Staubli VAL3: Control_Remote.pgx

public program Control_Remote(num& x_nMode, num& x_nCycleCount)
  local string l_sItem[2]
  local num l_nNum
  local num l_nKey
  local num l_nData[2]
  local num l_nSelectIndex
  local string l_sSMess[6]
begin

  //修改点位的 joint
  l_nData[0]=max(round(x_nMode),0)
  l_nData[1]=max(round(x_nCycleCount),0)

  l_sSMess[0]="按钮触发单工位"
  l_sSMess[1]="按钮触发单周期"
  l_sSMess[2]="按钮触发多周期"
  l_sSMess[3]="无需按钮触发"
  l_sSMess[4]="按钮触发排队"
  l_sSMess[5]="用户自定义触发"


  l_sItem[0]="生产模式:"+l_sSMess[l_nData[0]]
  l_sItem[1]="周期次数:"+toString("",l_nData[1])


  call Control_BottomS(",,,,,,取消,确定")
  call Control_PanelXY(8,0,25,2)
  call Control_ListCls()
  call Control_Panel("生产配置")
  call Control_List(l_sItem,l_nSelectIndex)
  while true
    l_nKey=getKey()

    switch l_nKey
      case 261
        l_nSelectIndex=max(0,l_nSelectIndex-1)
      break

      case 266
        l_nSelectIndex=min(l_nSelectIndex+1,1)
      break

      case 278
        x_nMode=l_nData[0]
        x_nCycleCount=l_nData[1]

        return
      break


      case 277
        return
      break

      case 270
        if l_nSelectIndex==0
         call Sel_Edit(l_nData[0],nPanelLTopX+10,nPanelLTopY+1,l_sSMess)
        else
          call Float_Edit(l_nData[1],nPanelLTopX+10,nPanelLTopY+2)

        endIf



        l_nData[l_nSelectIndex]=max(round(l_nData[l_nSelectIndex]),0)
      break

    endSwitch

    if l_nKey!=-1
  l_sItem[0]="生产模式:"+l_sSMess[l_nData[0]]
  l_sItem[1]="周期次数:"+toString("",l_nData[1])
      call Control_List(l_sItem,l_nSelectIndex)

    endIf






  endWhile





end
